Staubli VAL3: TestPositionCal.pgx

program TestPositionCal()
begin
  call DeplacementInit()

  call Deplacementpion(9,13)
  call Deplacementpion(22,18)

  call Deplacementpion(13,22)
  call Pionperdu(18,0)

  call Deplacementpion(26,19)
  call Pionperdu(22,1)

  call DeplacementInit()

end
